		30: (*Spr.*)
			IF mcHeightMoveAbsolute.Done AND
				(mcScrewer1MoveRelative.Done OR NOT bOptionScrewingBackwardsInPushingPosition OR NOT bRun1) AND 	
				(mcScrewer2MoveRelative.Done OR NOT bOptionScrewingBackwardsInPushingPosition OR NOT bRun2) 	 			
			THEN	
				mcHeightMoveAbsolute.Execute					:=	FALSE;
				mcScrewer1MoveRelative.Execute					:=	FALSE;
				mcScrewer2MoveRelative.Execute					:=	FALSE;	
				iToPushingPositionCASE							:=	iToPushingPositionCASE	+	10;
			END_IF

		40:  (*Opcja - Dodatkowe zamknięcie chwytakiem przed zakręceniem *)
				IF bOptionCapPositioning AND sTool <> 'ksztaltowa/do kulek' AND sTool <> 'wbijajaca' THEN
					CASE iCloseGripperBeforeScrewingCASE OF
						0:
							bGripper1Actuator					:=	bRun1;
							bGripper2Actuator					:=	bRun2;
							iCloseGripperBeforeScrewingCASE		:=	iCloseGripperBeforeScrewingCASE	+10;
						10:	
							IF 	(tonGripper1Delay.Q OR NOT bRun1) AND 
								(tonGripper2Delay.Q OR NOT bRun2) 
							THEN					
								iCloseGripperBeforeScrewingCASE	:=	iCloseGripperBeforeScrewingCASE	+10;
							END_IF
						20:	
								bGripper1Actuator				:=	bGripper1Actuator	:=	FALSE;		
								iCloseGripperBeforeScrewingCASE	:=	iCloseGripperBeforeScrewingCASE	+10;
						30:
							IF 	(tonGripper1ReliseDelay2.Q OR NOT bRun1) AND 
								(tonGripper2ReliseDelay2.Q OR NOT bRun2) 
							THEN					
								iCloseGripperBeforeScrewingCASE	:=	iCloseGripperBeforeScrewingCASE	+10;
							END_IF
						40:
						
							iCloseGripperBeforeScrewingCASE		:=	0;
							iToPushingPositionCASE				:=	iToPushingPositionCASE	+	10;							
					END_CASE
				ELSE
					iToPushingPositionCASE						:=	iToPushingPositionCASE	+	10;
				END_IF

			
		50:	 (*Zamkniecie chwytaka i przejazd dalej*)
			IF sTool <> 'ksztaltowa/do kulek' AND sTool <> 'wbijajaca' THEN
				bGripper1Actuator								:=	bRun1;
				bGripper2Actuator								:=	bRun2;
			ELSE                                    	
				bGripper1Actuator								:=	FALSE;
				bGripper2Actuator								:=	FALSE;
			END_IF	

			IF bOptionOpenedGripperWhenFindingScrew AND bOptionFindScrewInPushingPosition THEN
				bGripper1Actuator								:=	FALSE;
				bGripper2Actuator								:=	FALSE;
			END_IF
			
			IF 	(tonGripper1Delay.Q OR sTool = 'ksztaltowa/do kulek' OR sTool = 'wbijajaca' OR bOptionOpenedGripperWhenFindingScrew AND bOptionFindScrewInPushingPosition OR NOT bRun1) AND 
				(tonGripper2Delay.Q OR sTool = 'ksztaltowa/do kulek' OR sTool = 'wbijajaca' OR bOptionOpenedGripperWhenFindingScrew AND bOptionFindScrewInPushingPosition OR NOT bRun2) 
			THEN
          		         	
				iToPushingPositionCASE							:=	iToPushingPositionCASE	+	10;
			END_IF	
		
				
		60:(*Opcja - Obrót z pozycji docisku do zakrecania *)
			IF bOptionFindScrewRotateFromPushingToScrewingSensor AND NOT bOptionFindScrewInPushingPosition THEN
				lrFindigScrewDegree								:=	180;	
			                                    				
				uiScrewing1TorqueControl						:=	6000;
				mcScrewer1MoveRelative.Velocity					:=	lrScrewerSpeed;		
				mcScrewer1MoveRelative.Execute					:=	bRun1;
							                    				
				uiScrewing2TorqueControl						:=	6000;
				mcScrewer2MoveRelative.Velocity					:=	lrScrewerSpeed;		
				mcScrewer2MoveRelative.Execute					:=	bRun2;
				iToPushingPositionCASE							:=	iToPushingPositionCASE	+	10;
				
			ELSE 
				iToPushingPositionCASE							:=	iToPushingPositionCASE	+	10;
			END_IF
				
		70:
		
			IF bOptionFindScrewInPushingPosition THEN
				eRunningState									:=	E_GripperScrewer.eFindingScrew;
			ELSE
				eRunningState									:=	E_GripperScrewer.eToScrewingPosition;
			END_IF
			
			iToPushingPositionCASE						:=	0;
	
				
		END_CASE
		
		(*w1
		bGripper1Actuator								:=	FALSE;
		bGripper2Actuator								:=	FALSE;
		mcHeightMoveAbsolute.Execute					:=	TRUE;
		mcHeightMoveAbsolute.Velocity					:=	lrHeightSpeed;
		mcHeightMoveAbsolute.Position					:=	lrHeightPushingPosition;

		(*Opcja - obrót do tyłu w momencie dojazdu do pozycji docisku*)
		IF bOptionScrewingBackwardsInPushingPosition THEN
			lrFindigScrewDegree				:=	180;	
			
			uiScrewing1TorqueControl		:=	6000;
			mcScrewer1MoveRelative.Velocity	:=	lrScrewerSpeed/2;		
			mcScrewer1MoveRelative.Execute	:=	bRun1;
			
			uiScrewing2TorqueControl		:=	6000;
			mcScrewer2MoveRelative.Velocity	:=	lrScrewerSpeed/2;		
			mcScrewer2MoveRelative.Execute	:=	bRun2;
		END_IF
	
		IF mcHeightMoveAbsolute.Done AND
			(mcScrewer1MoveRelative.Done OR NOT bOptionScrewingBackwardsInPushingPosition OR NOT bRun1) AND // Opcja
			(mcScrewer2MoveRelative.Done OR NOT bOptionScrewingBackwardsInPushingPosition OR NOT bRun2) 	 // Opcja			
		THEN		
			
			IF bOptionCapPositioning THEN //OPCJA. Dodatkowe zamknięcie chwytakiem przed zakręceniem (do testów)
				CASE iCloseGripperBeforeScrewingCASE OF
					0:
						IF iTool <> 2 THEN
							bGripper1Actuator						:=	bRun1;
							bGripper2Actuator						:=	bRun2;
						ELSE
							bGripper1Actuator						:=	FALSE;
							bGripper2Actuator						:=	FALSE;
						END_IF
						
						iCloseGripperBeforeScrewingCASE		:=	iCloseGripperBeforeScrewingCASE	+10;
						
					10:	
						IF iTool <> 2 THEN
							bGripper1Actuator						:=	bRun1;
							bGripper2Actuator						:=	bRun2;
						ELSE
							bGripper1Actuator						:=	FALSE;
							bGripper2Actuator						:=	FALSE;
						END_IF		
							
						IF (tonGripper1Delay.Q OR NOT bRun1) AND (tonGripper2Delay.Q OR NOT bRun2) THEN
							bGripper1Actuator						:=	bGripper1Actuator	:=	FALSE;							
							iCloseGripperBeforeScrewingCASE	:=	iCloseGripperBeforeScrewingCASE	+10;
						END_IF
					
					20:
						IF  tonGripper1ReliseDelay.Q AND tonGripper2ReliseDelay.Q THEN // Czas na otwarcie chwytaków
											
							mcHeightMoveAbsolute.Execute			:=	FALSE;
							eRunningState							:=	E_GripperScrewer.eToScrewingPosition;
							iCloseGripperBeforeScrewingCASE	:=	0;
						END_IF
													
				END_CASE

			ELSE
				IF iTool <> 2 THEN
					bGripper1Actuator					:=	bRun1;
					bGripper2Actuator					:=	bRun2;
				ELSE
					bGripper1Actuator					:=	FALSE;
					bGripper2Actuator					:=	FALSE;
				END_IF
									
				IF ((tonGripper1Delay.Q OR NOT bRun1) AND (tonGripper2Delay.Q OR NOT bRun2)) OR bOptionOpenedGripperWhenFindingScrew THEN
					mcHeightMoveAbsolute.Execute		:=	FALSE;
					mcScrewer1MoveRelative.Execute		:=	FALSE;
					mcScrewer2MoveRelative.Execute		:=	FALSE;
					
					IF bOptionFindScrewRotateFromPushingToScrewingSensor THEN
						lrFindigScrewDegree				:=	180;	
			
						uiScrewing1TorqueControl		:=	6000;
						mcScrewer1MoveRelative.Velocity	:=	lrScrewerSpeed;		
						mcScrewer1MoveRelative.Execute	:=	bRun1;
						
						uiScrewing2TorqueControl		:=	6000;
						mcScrewer2MoveRelative.Velocity	:=	lrScrewerSpeed;		
						mcScrewer2MoveRelative.Execute	:=	bRun2;
					END_IF
					
					IF	(mcScrewer1MoveRelative.Execute OR NOT bRun1 OR NOT bOptionFindScrewRotateFromPushingToScrewingSensor) AND
						(mcScrewer2MoveRelative.Execute OR NOT bRun2 OR NOT bOptionFindScrewRotateFromPushingToScrewingSensor) THEN
						eRunningState						:=	E_GripperScrewer.eToScrewingPosition;
					END_IF
					IF bOptionFindScrewInPushingPosition AND NOT bOptionFindScrewRotateFromPushingToScrewingSensor THEN //Opcja - szukanie gwintu w pozycji docisku
						IF 	bOptionOpenedGripperWhenFindingScrew THEN //Opcja - szukanie gwintu na otwartym chwytaku
							bGripper1Actuator				:=	FALSE;
							bGripper2Actuator				:=	FALSE;
						END_IF					
					
						eRunningState					:=	E_GripperScrewer.eFindingScrew;
					END_IF
					
				END_IF	
			END_IF
		END_IF
	*)
END_ACTION

ACTION Running5FindingScrew:
(*Opcja 1 Szukania gwintu - zwykłe szukanie*) 
IF NOT bOptionFindScrewWithHeightSensor THEN
	(*Opcja cofniecie o zadany kąt*)	
	CASE iFindingScrewCASE OF
				
			0:	// Czyszczenie
				mcScrewer1MoveRelative.Execute				:=	FALSE;
				mcScrewer2MoveRelative.Execute				:=	FALSE;		
				lrScrewer1MaxTorqueWhenFindingScrew			:=	0;
				lrScrewer2MaxTorqueWhenFindingScrew			:=	0;
				lrStartPosition1FindingScrew 				:=	Screwing1AxisRef.NcToPlc.ActPos;
				lrStartPosition2FindingScrew 				:=	Screwing2AxisRef.NcToPlc.ActPos;			
				uiScrewing1TorqueControl					:=	6000;
				uiScrewing2TorqueControl					:=	6000;			
				bScrew1Found								:=	FALSE;
				bScrew2Found								:=	FALSE;
				iFindingScrewCASE							:=	iFindingScrewCASE	+	10;
						
			10: (*ruch o zadany kat*)
				mcScrewer1MoveRelative.Velocity		:=	lrScrewerSpeed;
				mcScrewer1MoveRelative.Execute		:=	bRun1;
				
				mcScrewer2MoveRelative.Velocity		:=	lrScrewerSpeed;
				mcScrewer2MoveRelative.Execute		:=	bRun2;
				
				IF	(NOT bRun1 OR mcScrewer1MoveRelative.Done) AND
					(NOT bRun2 OR mcScrewer2MoveRelative.Done)
			
				THEN		
					lrScrewer1MaxTorqueWhenFindingScrew	:= 0;
					lrScrewer2MaxTorqueWhenFindingScrew	:= 0;
					mcScrewer1MoveRelative.Execute		:=	FALSE;
					mcScrewer1MoveRelative.Execute		:=	FALSE;
					iFindingScrewCASE					:=	iFindingScrewCASE	+	10;	
				END_IF
					
			20:
				lrStartPosition1						:=	Screwing1AxisRef.NcToPlc.ActPos;
				lrStartPosition2						:=	Screwing2AxisRef.NcToPlc.ActPos;
				iFindingScrewCASE 						:=	0;
				eRunningState							:=	E_GripperScrewer.eScrewing;
				IF bOptionFindScrewInPushingPosition THEN // Opcja - szukanie gwintu w pozycji docisku
					// Przejście do pozycji zakręcania, dlatego że był w pozycji docisku
					eRunningState							:=	E_GripperScrewer.eToScrewingPosition;
				END_IF
				IF NOT bHeightGearingWithScrewer THEN 	(* Wersja bez gearowania*)
					mcScrewer1MoveVelocity.Execute		:= bRun1;
					mcScrewer2MoveVelocity.Execute		:= bRun2;
					eRunningState:=E_GripperScrewer.eScrewing;
				ELSE 									(* Wersja z gearowaniem*)
					iFindingScrewCASE 						:=	0;
					eRunningState							:=	E_GripperScrewer.eScrewing;
					IF bOptionFindScrewInPushingPosition THEN // Opcja - szukanie gwintu w pozycji docisku
						// Przejście do pozycji zakręcania, dlatego że był w pozycji docisku
						eRunningState							:=	E_GripperScrewer.eToScrewingPosition;
					END_IF
				END_IF
	END_CASE

ELSE (*Opcja 2 Szukania gwintu - szukanie z czujnikiem wysokości*) 
		CASE iFindingScrewCASE OF
			
		0:	// Czyszczenie
			mcScrewer1MoveRelative.Execute				:=	FALSE;
			lrStartPosition1FindingScrew 				:=	Screwing1AxisRef.NcToPlc.ActPos;
			lrStartPosition2FindingScrew 				:=	Screwing2AxisRef.NcToPlc.ActPos;			
			uiScrewing1TorqueControl					:=	6000;
			uiScrewing2TorqueControl					:=	6000;			
			bScrew1Found								:=	FALSE;
			bScrew2Found								:=	FALSE;
			bScrew1MinFound								:=	FALSE;
			bScrew2MinFound								:=	FALSE;			
			lrScrewerMaxSensorHeightWhenFindingScrew	:=	-100000;
			lrScrewerMinSensorHeightWhenFindingScrew	:=	100000;
			iFindingScrewCASE							:=	iFindingScrewCASE	+	10;


		

			
		10: // Rozpoczęcie ruchu w tył i szukanie MAX wysokości oraz uskoku - początek gwintu
			


			uiScrewing1TorqueControl					:=	6000;
			mcScrewer1MoveRelative.Velocity				:=	lrScrewerSpeed;
			//Zabezpieczenie - jak za szybko się kręci to nie opada zakręcarka i nie łapie gwintu
			IF mcScrewer1MoveRelative.Velocity > 2400	THEN
				mcScrewer1MoveRelative.Velocity			:= 2400;
			END_IF	
			mcScrewer1MoveRelative.Execute				:=	bRun1;				
			IF lrScrewerMaxSensorHeightWhenFindingScrew<rSensorHeightCV  THEN
				lrScrewerMaxSensorHeightWhenFindingScrew:=	rSensorHeightCV;
			END_IF			
			//Jak znajdziemy uskok - to początek gwintu - uskok o 0.3 do 0.5 podziałki bo całego nie wykryje
			IF ((rSensorHeightCV+lrPackageThreadPitch*0.3)<lrScrewerMaxSensorHeightWhenFindingScrew) THEN //Było z krotnoscia gwintu ale tak ma wiekszy sens
				bScrew1Found							:=	TRUE;
				lrStartPosition1FindingScrew 			:=	Screwing1AxisRef.NcToPlc.ActPos; //Pozycja złapania gwintu
			END_IF
			//Koniec wyszukiwania - albo koniec ruchu albo znaleziony gwint
			IF (mcScrewer1MoveRelative.Done OR NOT bRun1) OR bScrew1Found THEN
				mcScrewer1MoveRelative.Execute			:=	FALSE;
				mcScrewer1Stop.Execute					:= TRUE;
			//	bFindScrewAdjustSensorHeight			:=	FALSE;	
			//	iFindScrewAdjustSensorHeight			:=	iFindScrewAdjustSensorHeight	+	1;
					
				iFindingScrewCASE						:=	iFindingScrewCASE	+	10;
			END_IF

			
		20: // Przejście dalej gdy jest gotowość
			IF NOT mcScrewer1MoveRelative.Busy AND NOT mcScrewer2MoveRelative.Busy AND mcScrewer1Stop.Done THEN
				mcScrewer1Stop.Execute					:= 	FALSE;			
				iFindingScrewCASE						:=	iFindingScrewCASE	+	10;	
			END_IF
			
		30://Koniec ruchu
			lrStartPosition1						:=	lrStartPosition1FindingScrew;
			lrStartPosition2						:=	Screwing2AxisRef.NcToPlc.ActPos;
			iFindingScrewCASE 						:=	0;
			eRunningState							:=	E_GripperScrewer.eScrewing;
			IF bOptionFindScrewInPushingPosition THEN // Opcja - szukanie gwintu w pozycji docisku
				// Przejście do pozycji zakręcania, dlatego że był w pozycji docisku
				eRunningState							:=	E_GripperScrewer.eToScrewingPosition;
			END_IF
		END_CASE	
			
//		10: // Rozpoczęcie ruchu w tył i szukanie MIN i MAX momentu
//			// Tylko 1 zakręcarka szuka Min i Max po każdej zmianie
//			// Uruchom szukanie jeżeli są wartości domyślne
//			IF lrScrewerMaxSensorHeightWhenFindingScrew = -100000 OR lrScrewerMinSensorHeightWhenFindingScrew = 100000 THEN
//				bFindScrewAdjustSensorHeight				:= TRUE;
//				lrScrewerMaxSensorHeightWhenFindingScrew	:=	-100000; //Musi być INIT -100000
//				lrScrewerMinSensorHeightWhenFindingScrew	:=	100000;
//			END_IF
			
//			IF bFindScrewAdjustSensorHeight THEN
//				uiScrewing1TorqueControl					:=	6000;
//				lrFindigScrewDegree							:=	720;
//				mcScrewer1MoveRelative.Velocity				:=	200;
//				mcScrewer1MoveRelative.Execute				:=	bRun1;
							
//				IF lrScrewerMaxSensorHeightWhenFindingScrew<diSensorHeightCV THEN
//					lrScrewerMaxSensorHeightWhenFindingScrew:=	diSensorHeightCV;
//				END_IF			
//				IF lrScrewerMinSensorHeightWhenFindingScrew>diSensorHeightCV THEN
//					lrScrewerMinSensorHeightWhenFindingScrew:=	diSensorHeightCV;
//				END_IF		
			
//				IF (mcScrewer1MoveRelative.Done OR NOT bRun1) THEN
//					mcScrewer1MoveRelative.Execute			:=	FALSE;
//					bFindScrewAdjustSensorHeight			:=	FALSE;	iFindScrewAdjustSensorHeight	:=	iFindScrewAdjustSensorHeight	+	1;
//					iFindingScrewCASE						:=	iFindingScrewCASE	+	10;
//				END_IF
//			ELSE
//				iFindingScrewCASE						:=	iFindingScrewCASE	+	10;
//			END_IF

			
//		30: // Rozpoczęcie szukanie największego momentu o określony maksymalny kąt
//			uiScrewing1TorqueControl					:=	6000;
//			mcScrewer1MoveRelative.Velocity				:=	500;//lrScrewerSpeed;///2;
//			mcScrewer1MoveRelative.Execute				:=	bRun1;
			
//			uiScrewing2TorqueControl					:=	6000;
//			mcScrewer2MoveRelative.Velocity				:=	500;//lrScrewerSpeed;///2;
//			mcScrewer2MoveRelative.Execute				:=	bRun2;		
	
//			iFindingScrewCASE							:=	iFindingScrewCASE	+	10;	
			
//		40:	//Szukanie określonego momentu po 200 st. i zatrzymanie ruchu 


//			(*Pierwsze szukanie*)
//			IF NOT bScrew1MinFound THEN															(*W1*)
//				IF ABS(ABS(lrStartPosition1FindingScrew)-ABS(Screwing1AxisRef.NcToPlc.ActPos))	>	100  THEN 
//					//IF lrScrewer1ActualTorque > (lrScrewer1MinTorqueWhenFindingScrew - 5) AND lrScrewer1ActualTorque < (lrScrewer1MaxTorqueWhenFindingScrew + 15) THEN		
////					IF diSensorHeightCV < -39000 THEN		(*W2*) //Dla Słoików 300ml
//					IF diSensorHeightCV < ((lrScrewerMaxSensorHeightWhenFindingScrew+lrScrewerMinSensorHeightWhenFindingScrew)/2) THEN		(*W2*) //Dla Słoików 300ml						
//						bScrew1MinFound						:=	TRUE;
//						lrStartPosition1FindingScrew 		:=	Screwing1AxisRef.NcToPlc.ActPos;
//					END_IF	
//				END_IF
//			END_IF
//			IF NOT bScrew2MinFound THEN															(*W1*)
//				IF ABS(ABS(lrStartPosition2FindingScrew)-ABS(Screwing2AxisRef.NcToPlc.ActPos))	>	100  THEN 
////					IF diSensorHeightCV < -39000 THEN		(*W2*)	//Dla Słoików 300ml	
//					IF diSensorHeightCV < ((lrScrewerMaxSensorHeightWhenFindingScrew+lrScrewerMinSensorHeightWhenFindingScrew)/2) THEN		(*W2*)	//Dla Słoików 300ml	
//						bScrew2MinFound						:=	TRUE;	
//						lrStartPosition2FindingScrew 		:=	Screwing2AxisRef.NcToPlc.ActPos;
//					END_IF	
//				END_IF	
//			END_IF
//			lrScrewerOffsetSensorHeightWhenFindingScrew	:=	((lrScrewerMaxSensorHeightWhenFindingScrew+lrScrewerMinSensorHeightWhenFindingScrew)/2)
//																+(lrScrewerMinSensorHeightWhenFindingScrew-lrScrewerMaxSensorHeightWhenFindingScrew)/6;
			
//			(*Drugie szukanie*)																					(*W3*)
//			IF bScrew1MinFound AND ABS(ABS(lrStartPosition1FindingScrew)-ABS(Screwing1AxisRef.NcToPlc.ActPos))	>	10  THEN 
				
//				IF diSensorHeightCV > lrScrewerOffsetSensorHeightWhenFindingScrew THEN		(*W4*)	//Dla Słoików 300ml
//					bScrew1Found						:=	TRUE;
//					mcScrewer1MoveRelative.Execute		:=	FALSE;
//					lrStartPosition1FindingScrew 		:=	Screwing1AxisRef.NcToPlc.ActPos;
//				END_IF
//			END_IF																								(*W3*)
//			IF bScrew2MinFound AND ABS(ABS(lrStartPosition2FindingScrew)-ABS(Screwing2AxisRef.NcToPlc.ActPos))	>	10  THEN 
//				IF diSensorHeightCV > ((lrScrewerMaxSensorHeightWhenFindingScrew+lrScrewerMinSensorHeightWhenFindingScrew)/2) THEN		(*W4*)	//Dla Słoików 300ml
//					bScrew2Found						:=	TRUE;
//					mcScrewer2MoveRelative.Execute		:=	FALSE;
//					lrStartPosition2FindingScrew 		:=	Screwing1AxisRef.NcToPlc.ActPos;
//				END_IF
//			END_IF

//			IF bScrew1Found  THEN

//				uiScrewing1TorqueControl		:=	6000;
//				mcScrewer1Stop.Execute			:=	TRUE;
				
//			END_IF
			
//			IF bScrew2Found  THEN

//				uiScrewing2TorqueControl		:=	6000;
//				mcScrewer2Stop.Execute			:=	TRUE;
//			END_IF			
			
//			IF	((bScrew1Found AND mcScrewer1Stop.Done) OR NOT bRun1 OR mcScrewer1MoveRelative.Done) AND
//				((bScrew2Found AND mcScrewer2Stop.Done) OR NOT bRun2 OR mcScrewer2MoveRelative.Done)
//			THEN
//				 mcScrewer1MoveRelative.Execute 	:=	FALSE;
//				 mcScrewer1Stop.Execute				:=	FALSE;
//				 mcScrewer2MoveRelative.Execute 	:=	FALSE;		
//				 mcScrewer2Stop.Execute				:=	FALSE;	 
//				 iFindingScrewCASE					:=	iFindingScrewCASE	+	10;	
//			END_IF
			
//		50: 
//			IF tonFindingScrewDelay.Q THEN
// 				iFindingScrewCASE					:=	iFindingScrewCASE	+	10;						
//			END_IF




END_IF
END_ACTION

ACTION Running6ScrewingMomentaryMode:
IF mcScrewer1TorqueControl.Error OR mcScrewer1MoveVelocity.Error OR mcScrewer1MoveVelocity2.Error
	 OR mcScrewer1MoveVelocity3.Error OR mcScrewer1MoveRelative.Error OR mcScrewer1MoveAbsolute.Error THEN
	bTest:= TRUE;
END_IF
tonInEndVelocity(IN:=mcScrewer1MoveContinuousRel.InEndVelocity, PT:=T#2MS);


				(********** TRYB MOMENTOWY **********)
					CASE iScrewingCase OF 	
					0:
						(* Wersja 2 - gearowanie Multi Master***************************************************************) 
						IF iTool <> 2 THEN
							bGripper1Actuator						:=	bRun1; // Ponowne załączanie chwytaków, dlatego
							bGripper2Actuator						:=	bRun2; // że jest możliwa duża ilość opcji
						ELSE
							bGripper1Actuator						:=	FALSE; // Ponowne załączanie chwytaków, dlatego
							bGripper2Actuator						:=	FALSE;
						END_IF
						//Właczenie sięcia osi
						mcHeightGearInMultiMaster.Enable			:=	TRUE;				
						//Jak osie spięte to początek kręcenia
						IF	mcHeightGearInMultiMaster.InGear AND 
							(tonGripper1Delay.Q OR sTool = 'ksztaltowa/do kulek' OR NOT bRun1) AND (tonGripper2Delay.Q OR sTool = 'ksztaltowa/do kulek'  OR NOT bRun2) // ton'y powinny być już wczesniej załączone jeżeli były chwytaki	
						THEN
							//Bloczek obrotu o zadany kąt i kontynuowania ruchu z zadaną prędkością
							mcScrewer1MoveContinuousRel.Execute				:= bRun1;
							//Kąt zmodyfikowany o różnicę między pozycją zatrzymania zakręcarki a pozycją wykrycia gwintu
							mcScrewer1MoveContinuousRel.Distance			:= Screwing1AxisRef.NcToPlc.ActPos - lrStartPosition1 + lrPackageTurnoversToFullScrewed*360.0-30.0;

							//DODAĆ ZABEZPIECZENIE JAK WYJDZIE ABSURDALNY KĄT
							
							//Prędkość na wyjściu z bloczka 120RPM - Inercja zakręcarki jest rozsądna
							mcScrewer1MoveContinuousRel.EndVelocity			:= 360*2;
							//Prędkość zakręcania wg parametrów
							mcScrewer1MoveContinuousRel.Velocity			:= (lrScrewerSpeed);
														
							iScrewingCase									:=	25;//iScrewingCase + 10;			
						END_IF
						
					10:	
					
						IF ABS(ABS(lrStartPosition1)-ABS(Screwing1AxisRef.NcToPlc.ActPos))>(lrPackageTurnoversToFullScrewed*360.0-90.0)  THEN 
							mcScrewer1MoveVelocity.Execute					:= FALSE;
							mcScrewer1MoveVelocity2.Execute					:= bRun1;
							mcScrewer1MoveVelocity2.Velocity				:= 360;
							uiScrewing1TorqueControl						:=	60000;
						//	mcScrewer1TorqueControl.Torque					:=	-5000;		
						//	mcScrewer1TorqueControl.TorqueRamp				:=	80000;	
							mcScrewer1TorqueControl.VelocityLimitHigh		:=	360;//(lrScrewerSpeed)/3.0;
							mcScrewer1TorqueControl.VelocityLimitLow		:=	-360;//-(lrScrewerSpeed)/3.0;
							iScrewingCase									:=	iScrewingCase + 10;	
						END_IF	
							
//						IF ABS(ABS(lrStartPosition2)-ABS(Screwing2AxisRef.NcToPlc.ActPos))>(lrPackageTurnoversToFullScrewed*360.0/7)  THEN 
//							mcScrewer2TorqueControl.Torque					:=	-9;		
//							mcScrewer2TorqueControl.TorqueRamp				:=	1500;					
//							mcScrewer2TorqueControl.VelocityLimitLow		:=	-4000;
//						END_IF	
					20:	
						mcScrewer1MoveVelocity2.Execute					:= FALSE;
						IF ABS(ABS(lrStartPosition1)-ABS(Screwing1AxisRef.NcToPlc.ActPos))>(lrPackageTurnoversToFullScrewed*360.0-15.0)  THEN
							mcScrewer1MoveVelocity2.Execute					:= FALSE;
							mcScrewer1TorqueControl.Execute					:=	bRun1;
							mcScrewer1TorqueControl.Torque					:=	(INT_TO_UINT(iScrewer1SetTorque)+iScrewer1AddTorque);		
						//	mcScrewer1TorqueControl.TorqueRamp				:=	4000;					
						//	mcScrewer1TorqueControl.VelocityLimitLow		:=	- 10;//(lrScrewerSpeed)/3.0;
							iScrewingCase									:=	iScrewingCase + 10;	
						END_IF	
							
						IF ABS(ABS(lrStartPosition2)-ABS(Screwing2AxisRef.NcToPlc.ActPos))>(lrPackageTurnoversToFullScrewed*360.0/6)  THEN 
							mcScrewer2TorqueControl.Torque					:=	(INT_TO_UINT(iScrewer2SetTorque)+iScrewer2AddTorque);		
							mcScrewer2TorqueControl.TorqueRamp				:=	4000;					
							mcScrewer2TorqueControl.VelocityLimitLow		:=	-(lrScrewerSpeed);
						END_IF	
						
					25:
						//Jak dojedzie do końca ruchu
						IF mcScrewer1MoveContinuousRel.InEndVelocity AND tonInEndVelocity.Q THEN
							mcScrewer1MoveContinuousRel.Execute				:= FALSE;
							//Przygotowanie trybu momentowego
							mcScrewer1TorqueControl.Execute					:=	bRun1;
							mcScrewer1TorqueControl.Torque					:=	(INT_TO_UINT(iScrewer1SetTorque)+iScrewer1AddTorque);	
							mcScrewer1TorqueControl.TorqueRamp				:=	8000;
							mcScrewer1TorqueControl.VelocityLimitHigh		:=	360*2;//(lrScrewerSpeed)/3.0;
							mcScrewer1TorqueControl.VelocityLimitLow		:=	-360*2;//-(lrScrewerSpeed)/3.0;	
							iScrewingCase									:=	30;//iScrewingCase + 10;	
						END_IF
	
					30:
						IF tonMomentaryScrewing1Timer.Q OR bWarning1 THEN
							mcScrewer1Stop.Execute				:=	TRUE;
							bGripper1Actuator					:=	FALSE;
							mcScrewer1TorqueControl.Execute		:=	FALSE;
							uiScrewing1TorqueControl			:=	0;
							bScrewed1							:=	TRUE;	
						END_IF
						IF tonMomentaryScrewing2Timer.Q OR bWarning2 THEN
							mcScrewer2Stop.Execute				:=	TRUE;
							bGripper2Actuator					:=	FALSE;
							mcScrewer2TorqueControl.Execute		:=	FALSE;
							uiScrewing2TorqueControl			:=	0;
							bScrewed2							:=	TRUE;		
						END_IF
				
						// Warunki zakręcenia zaleznie od uruchomionej zakręcarki
						IF (bScrewed1 OR NOT bRun1) AND (bScrewed2 OR NOT bRun2) AND
							(mcScrewer1Stop.Done OR NOT mcScrewer1Stop.Execute) AND 
							(mcScrewer2Stop.Done OR NOT mcScrewer2Stop.Execute) THEN
								mcScrewer1Stop.Execute			:= FALSE;
								mcScrewer2Stop.Execute			:= FALSE;
								iScrewingCase					:= iScrewingCase + 10;		
						END_IF
					40:
						(* Rozgearowanie osi *)
						mcHeightGearOut.Execute				:=	TRUE;
						mcHeightGearInMultiMaster.Enable	:=	FALSE;
	
						IF  mcHeightGearOut.Done THEN
							mcHeightGearOut.Execute					:= FALSE;
							eRunningState							:= E_GripperScrewer.eHolding;	
							iScrewingCase							:= 0;	
						END_IF			
					END_CASE
END_ACTION

ACTION Running6ScrewingPositionTorqueMode:
				(********* TRYB POZYCYJNY  *********)
				
				lrPackageThreadPitch;	
				(*Wymuszanie zwiększonego momentu przez 1/4 całego zakręcania*)
				IF ABS(ABS(lrStartPosition1)-ABS(Screwing1AxisRef.NcToPlc.ActPos))>(lrPackageTurnoversToFullScrewed*360.0/7)  THEN 
							uiScrewing1TorqueControl			:=	(INT_TO_UINT(iScrewer1SetTorque+3)*10)+(iScrewer1AddTorque*10);	
				ELSE		uiScrewing1TorqueControl			:=	6000;
				END_IF
				//uiScrewing1TorqueControl			:=	(INT_TO_UINT(iScrewerSetTorque+3)*10)+iScrewer1AddTorque;	
				(*Wymuszanie zwiększonego momentu przez 1/4 całego zakręcania*)
				IF ABS(ABS(lrStartPosition2)-ABS(Screwing2AxisRef.NcToPlc.ActPos))>(lrPackageTurnoversToFullScrewed*360.0/7)  THEN 
							uiScrewing2TorqueControl			:=	(INT_TO_UINT(iScrewer2SetTorque+3)*10)+(iScrewer2AddTorque*10);		
				ELSE		uiScrewing2TorqueControl			:=	6000;
				END_IF	

					CASE iScrewingCase OF 	
					0:
						(* Wersja 2 - gearowanie Multi Master***************************************************************) 
						IF iTool <> 2 THEN
							bGripper1Actuator						:=	bRun1; // Ponowne załączanie chwytaków, dlatego
							bGripper2Actuator						:=	bRun2; // że jest możliwa duża ilość opcji
						ELSE
							bGripper1Actuator						:=	FALSE; // Ponowne załączanie chwytaków, dlatego
							bGripper2Actuator						:=	FALSE; // że jest możliwa duża ilość opcji
						END_IF
						mcHeightGearInMultiMaster.Enable			:=	TRUE;				
						(* Start zakręcania *)
						IF	mcHeightGearInMultiMaster.InGear AND 
							(tonGripper1Delay.Q OR sTool = 'ksztaltowa/do kulek' OR NOT bRun1) AND (tonGripper2Delay.Q OR sTool = 'ksztaltowa/do kulek' OR NOT bRun2) // ton'y powinny być już wczesniej załączone jeżeli były chwytaki	
						THEN

							CASE iScrewing2Case OF 	
								
							0:
							
								mcScrewer1MoveVelocity2.Velocity		:=	5000;
								mcScrewer1MoveVelocity2.Execute		:=	bRun1;
								mcScrewer1MoveVelocity2.Direction	:=	MC_Positive_Direction;
																				
								mcScrewer2MoveVelocity2.Velocity		:=	5000;
								mcScrewer2MoveVelocity2.Execute		:=	bRun2;
								mcScrewer2MoveVelocity2.Direction	:=	MC_Positive_Direction;	
	
								iScrewing2Case						:=	iScrewing2Case + 10;										
							
							10:
								mcScrewer1MoveVelocity2.Execute		:=	FALSE;
								mcScrewer2MoveVelocity2.Execute		:=	FALSE;
							
								iScrewing2Case						:=	iScrewing2Case + 10;
	
							20:
							
								mcScrewer1MoveVelocity.Velocity		:=	lrScrewerSpeed;		
								mcScrewer1MoveVelocity.Direction	:=	MC_Positive_Direction;	
								IF ABS(ABS(lrStartPosition1)-ABS(Screwing1AxisRef.NcToPlc.ActPos))>(lrPackageTurnoversToFullScrewed*360.0/7)  THEN 									
									mcScrewer1MoveVelocity.Execute		:=	bRun1;									
								END_IF
								mcScrewer2MoveVelocity.Velocity		:=	lrScrewerSpeed;	
								mcScrewer1MoveVelocity.Direction		:=	MC_Positive_Direction;	
								IF ABS(ABS(lrStartPosition2)-ABS(Screwing2AxisRef.NcToPlc.ActPos))>(lrPackageTurnoversToFullScrewed*360.0/7)  THEN 
	
									mcScrewer2MoveVelocity.Execute		:=	bRun2;
								END_IF			

								IF (mcScrewer1MoveVelocity.Execute OR NOT bRun1) AND (mcScrewer2MoveVelocity.Execute OR NOT bRun2) THEN
									iScrewing2Case					:= 0	;
									iScrewingCase					:= iScrewingCase + 10;		
								END_IF
								
							END_CASE
							
						END_IF
						
					10:	
					
						(*Zmniejszanie prędkości jeżeli jest już przytrzymanie*)
						IF tonTightScrewing1Timer.ET > T#0S AND Screwing1AxisRef.NcToPlc.ActVelo < 10 THEN
							//mcScrewer1MoveVelocity.Execute		:= FALSE;
							//mcScrewer1MoveVelocity2.Execute		:= FALSE;
							
							//mcScrewer1MoveVelocity3.Velocity	:=	10;
							//mcScrewer1MoveVelocity3.Execute		:=	bRun1;
							//mcScrewer1MoveVelocity3.Direction	:=	MC_Positive_Direction;		

							rScrewing1ProportionalGain	:= 0;
							//rScrewing2ProportionalGain	:= 0;												
						END_IF
						
						IF tonTightScrewing2Timer.ET > T#0S AND Screwing2AxisRef.NcToPlc.ActVelo < 10 THEN
							//mcScrewer2MoveVelocity.Execute		:= FALSE;
							//mcScrewer2MoveVelocity2.Execute		:= FALSE;
							
							//mcScrewer2MoveVelocity3.Velocity	:=	10;
							//mcScrewer2MoveVelocity3.Execute		:=	bRun1;
							//mcScrewer2MoveVelocity3.Direction	:=	MC_Positive_Direction;		

							//rScrewing1ProportionalGain	:= 0;
							rScrewing2ProportionalGain	:= 0;												
						END_IF					
					
						(* Sprawdzanie czy osiągnięto moment lub zbyt długie zakracanie*)				
						IF tonTightScrewing1Timer.Q OR bWarning1 THEN
							bGripper1Actuator					:=	FALSE;
							bScrewed1							:=	TRUE;	
						END_IF
						IF tonTightScrewing2Timer.Q OR bWarning2 THEN
							bGripper2Actuator					:=	FALSE;
							bScrewed2							:=	TRUE;		
						END_IF
	
						IF tonTightScrewing1TimerAndOpenedGripper.Q THEN
							mcScrewer1Stop.Execute				:=	TRUE;
							mcScrewer1MoveVelocity.Execute		:=	FALSE;
							mcScrewer1MoveVelocity2.Execute		:=	FALSE;
							mcScrewer1MoveVelocity3.Execute		:=	FALSE;							
							uiScrewing1TorqueControl			:=	0;
						END_IF
						IF tonTightScrewing2TimerAndOpenedGripper.Q THEN
							mcScrewer2Stop.Execute				:=	TRUE;
							mcScrewer2MoveVelocity.Execute		:=	FALSE;
							mcScrewer2MoveVelocity2.Execute		:=	FALSE;	
							mcScrewer2MoveVelocity3.Execute		:=	FALSE;							
							uiScrewing2TorqueControl			:=	0;
						END_IF
					
						// Warunki zakręcenia zaleznie od uruchomionej zakręcarki
						IF (tonTightScrewing1TimerAndOpenedGripper.Q OR NOT bRun1) AND (tonTightScrewing2TimerAndOpenedGripper.Q OR NOT bRun2) AND
							(mcScrewer1Stop.Done OR NOT mcScrewer1Stop.Execute) AND 
							(mcScrewer2Stop.Done OR NOT mcScrewer2Stop.Execute) THEN
								mcScrewer1Stop.Execute			:= FALSE;
								mcScrewer2Stop.Execute			:= FALSE;
								iScrewingCase					:= iScrewingCase + 10;		
						END_IF
						
					20:
						(* Rozgearowanie osi *)
						mcHeightGearOut.Execute				:=	TRUE;
						mcHeightGearInMultiMaster.Enable	:=	FALSE;
	
						IF  mcHeightGearOut.Done THEN
							mcHeightGearOut.Execute					:= FALSE;
							eRunningState							:= E_GripperScrewer.eHolding;	
							iScrewingCase							:= 0;	
						END_IF			
					END_CASE
END_ACTION

ACTION Screwer1ControlBlocks:
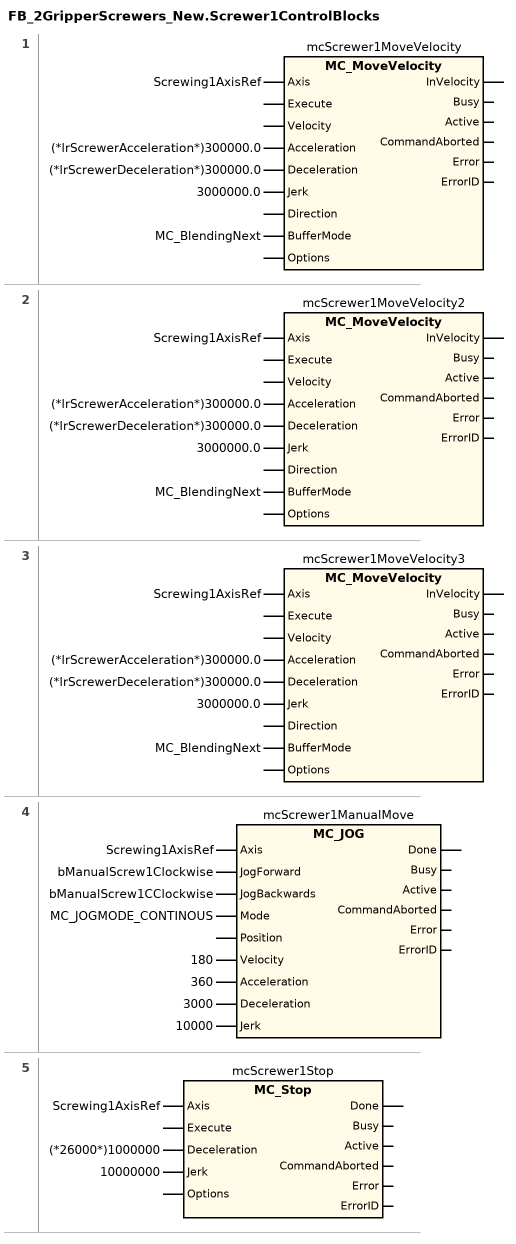
// NETWORK 1
mcScrewer1MoveVelocity(
    Axis := Screwing1AxisRef,
    Acceleration := (*lrScrewerAcceleration*)300000.0,
    Deceleration := (*lrScrewerDeceleration*)300000.0,
    Jerk := 3000000.0,
    BufferMode := MC_BlendingNext); // MC_MoveVelocity

// NETWORK 2
mcScrewer1MoveVelocity2(
    Axis := Screwing1AxisRef,
    Acceleration := (*lrScrewerAcceleration*)300000.0,
    Deceleration := (*lrScrewerDeceleration*)300000.0,
    Jerk := 3000000.0,
    BufferMode := MC_BlendingNext); // MC_MoveVelocity

// NETWORK 3
mcScrewer1MoveVelocity3(
    Axis := Screwing1AxisRef,
    Acceleration := (*lrScrewerAcceleration*)300000.0,
    Deceleration := (*lrScrewerDeceleration*)300000.0,
    Jerk := 3000000.0,
    BufferMode := MC_BlendingNext); // MC_MoveVelocity

// NETWORK 4
mcScrewer1ManualMove(
    Axis := Screwing1AxisRef,
    JogForward := bManualScrew1Clockwise,
    JogBackwards := bManualScrew1CClockwise,
    Mode := MC_JOGMODE_CONTINOUS,
    Velocity := 180,
    Acceleration := 360,
    Deceleration := 3000,
    Jerk := 10000); // MC_JOG

// NETWORK 5
mcScrewer1Stop(Axis := Screwing1AxisRef, Deceleration := (*26000*)1000000, Jerk := 10000000); // MC_Stop

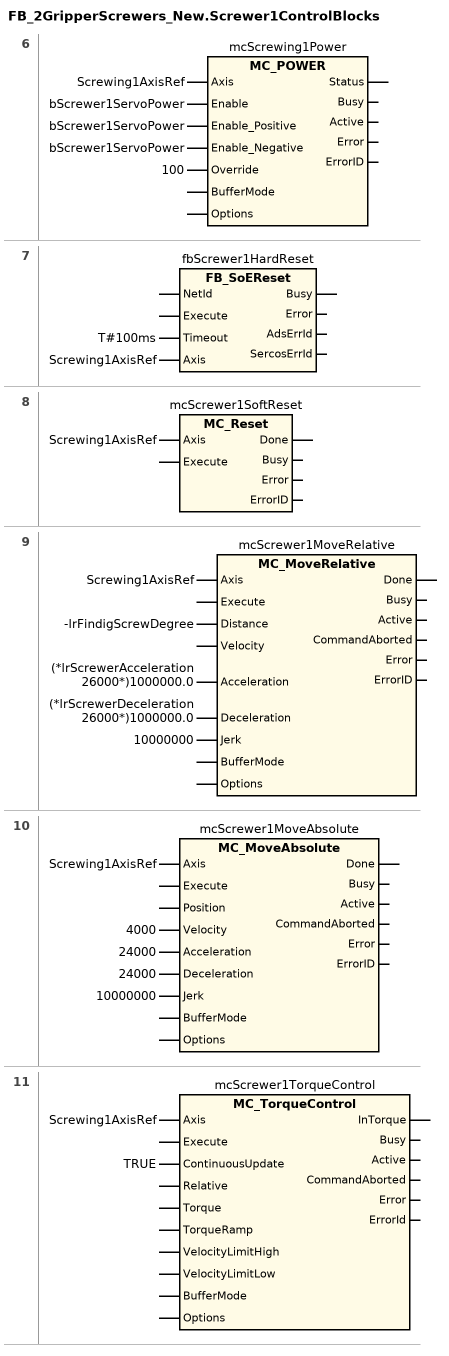
// NETWORK 6
mcScrewing1Power(
    Axis := Screwing1AxisRef,
    Enable := bScrewer1ServoPower,
    Enable_Positive := bScrewer1ServoPower,
    Enable_Negative := bScrewer1ServoPower,
    Override := 100); // MC_POWER

// NETWORK 7
fbScrewer1HardReset(Timeout := T#100ms, Axis := Screwing1AxisRef); // FB_SoEReset

// NETWORK 8
mcScrewer1SoftReset(Axis := Screwing1AxisRef); // MC_Reset

// NETWORK 9
mcScrewer1MoveRelative(
    Axis := Screwing1AxisRef,
    Distance := -lrFindigScrewDegree,
    Acceleration := (*lrScrewerAcceleration 26000*)1000000.0,
    Deceleration := (*lrScrewerDeceleration 26000*)1000000.0,
    Jerk := 10000000); // MC_MoveRelative

// NETWORK 10
mcScrewer1MoveAbsolute(
    Axis := Screwing1AxisRef,
    Velocity := 4000,
    Acceleration := 24000,
    Deceleration := 24000,
    Jerk := 10000000); // MC_MoveAbsolute

// NETWORK 11
mcScrewer1TorqueControl(Axis := Screwing1AxisRef, ContinuousUpdate := TRUE); // MC_TorqueControl

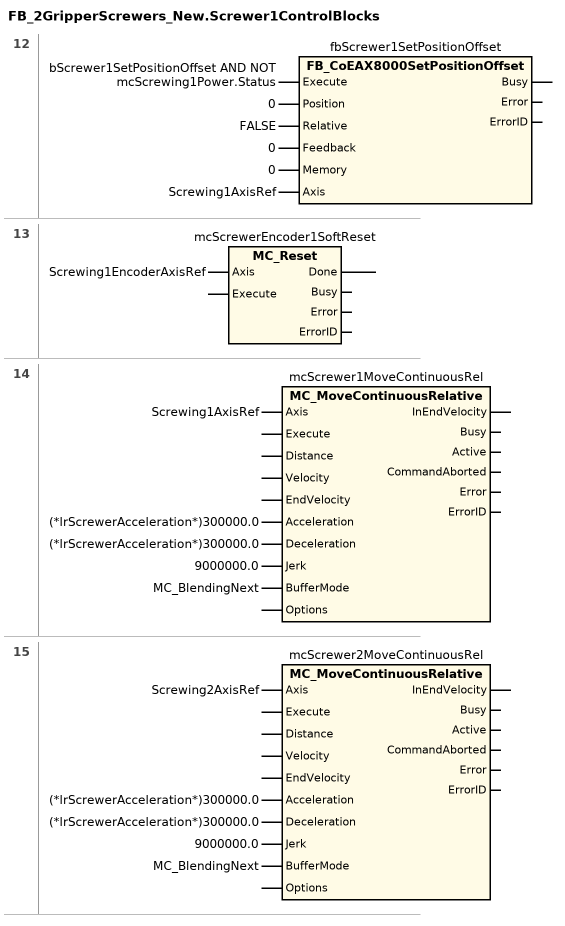
// NETWORK 12
fbScrewer1SetPositionOffset(
    Execute := bScrewer1SetPositionOffset AND NOT mcScrewing1Power.Status,
    Position := 0,
    Relative := FALSE,
    Feedback := 0,
    Memory := 0,
    Axis := Screwing1AxisRef); // FB_CoEAX8000SetPositionOffset

// NETWORK 13
mcScrewerEncoder1SoftReset(Axis := Screwing1EncoderAxisRef); // MC_Reset

// NETWORK 14
mcScrewer1MoveContinuousRel(
    Axis := Screwing1AxisRef,
    Acceleration := (*lrScrewerAcceleration*)300000.0,
    Deceleration := (*lrScrewerAcceleration*)300000.0,
    Jerk := 9000000.0,
    BufferMode := MC_BlendingNext); // MC_MoveContinuousRelative

// NETWORK 15
mcScrewer2MoveContinuousRel(
    Axis := Screwing2AxisRef,
    Acceleration := (*lrScrewerAcceleration*)300000.0,
    Deceleration := (*lrScrewerAcceleration*)300000.0,
    Jerk := 9000000.0,
    BufferMode := MC_BlendingNext); // MC_MoveContinuousRelative
END_ACTION

ACTION Screwer2ControlBlocks:
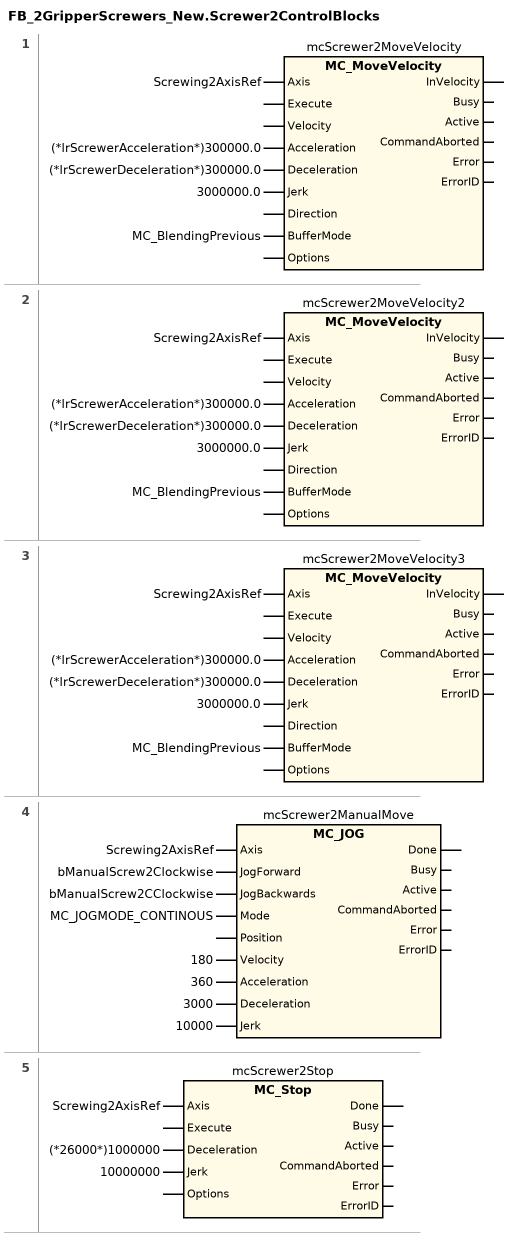
// NETWORK 1
mcScrewer2MoveVelocity(
    Axis := Screwing2AxisRef,
    Acceleration := (*lrScrewerAcceleration*)300000.0,
    Deceleration := (*lrScrewerDeceleration*)300000.0,
    Jerk := 3000000.0,
    BufferMode := MC_BlendingPrevious); // MC_MoveVelocity

// NETWORK 2
mcScrewer2MoveVelocity2(
    Axis := Screwing2AxisRef,
    Acceleration := (*lrScrewerAcceleration*)300000.0,
    Deceleration := (*lrScrewerDeceleration*)300000.0,
    Jerk := 3000000.0,
    BufferMode := MC_BlendingPrevious); // MC_MoveVelocity

// NETWORK 3
mcScrewer2MoveVelocity3(
    Axis := Screwing2AxisRef,
    Acceleration := (*lrScrewerAcceleration*)300000.0,
    Deceleration := (*lrScrewerDeceleration*)300000.0,
    Jerk := 3000000.0,
    BufferMode := MC_BlendingPrevious); // MC_MoveVelocity

// NETWORK 4
mcScrewer2ManualMove(
    Axis := Screwing2AxisRef,
    JogForward := bManualScrew2Clockwise,
    JogBackwards := bManualScrew2CClockwise,
    Mode := MC_JOGMODE_CONTINOUS,
    Velocity := 180,
    Acceleration := 360,
    Deceleration := 3000,
    Jerk := 10000); // MC_JOG

// NETWORK 5
mcScrewer2Stop(Axis := Screwing2AxisRef, Deceleration := (*26000*)1000000, Jerk := 10000000); // MC_Stop

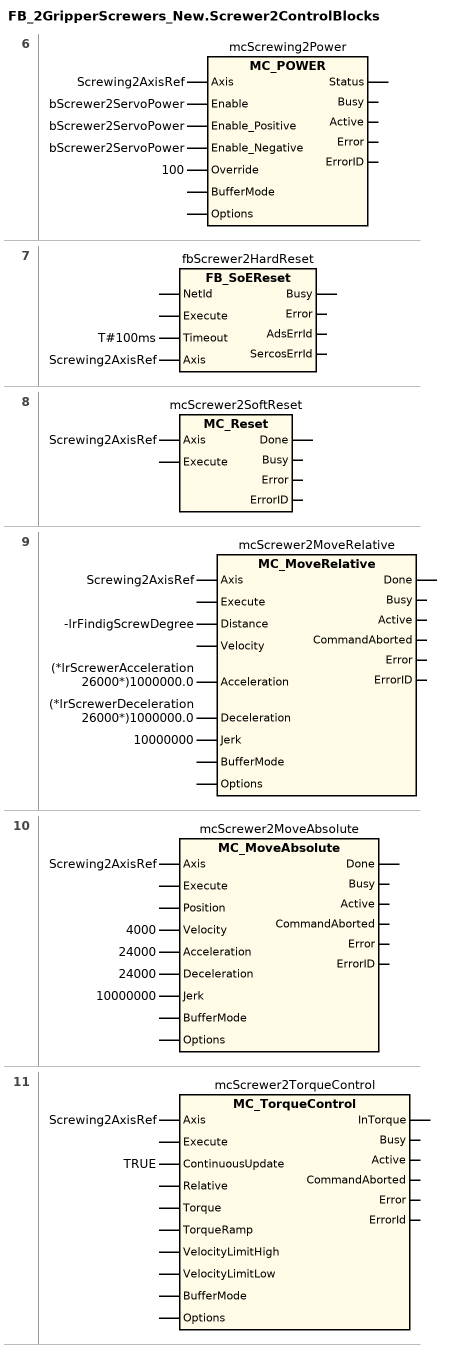
// NETWORK 6
mcScrewing2Power(
    Axis := Screwing2AxisRef,
    Enable := bScrewer2ServoPower,
    Enable_Positive := bScrewer2ServoPower,
    Enable_Negative := bScrewer2ServoPower,
    Override := 100); // MC_POWER

// NETWORK 7
fbScrewer2HardReset(Timeout := T#100ms, Axis := Screwing2AxisRef); // FB_SoEReset

// NETWORK 8
mcScrewer2SoftReset(Axis := Screwing2AxisRef); // MC_Reset

// NETWORK 9
mcScrewer2MoveRelative(
    Axis := Screwing2AxisRef,
    Distance := -lrFindigScrewDegree,
    Acceleration := (*lrScrewerAcceleration 26000*)1000000.0,
    Deceleration := (*lrScrewerDeceleration 26000*)1000000.0,
    Jerk := 10000000); // MC_MoveRelative

// NETWORK 10
mcScrewer2MoveAbsolute(
    Axis := Screwing2AxisRef,
    Velocity := 4000,
    Acceleration := 24000,
    Deceleration := 24000,
    Jerk := 10000000); // MC_MoveAbsolute

// NETWORK 11
mcScrewer2TorqueControl(Axis := Screwing2AxisRef, ContinuousUpdate := TRUE); // MC_TorqueControl

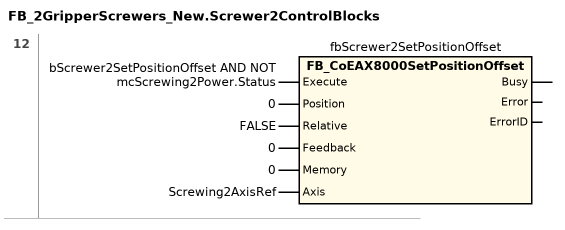
// NETWORK 12
fbScrewer2SetPositionOffset(
    Execute := bScrewer2SetPositionOffset AND NOT mcScrewing2Power.Status,
    Position := 0,
    Relative := FALSE,
    Feedback := 0,
    Memory := 0,
    Axis := Screwing2AxisRef); // FB_CoEAX8000SetPositionOffset
END_ACTION

ACTION Simulation:
(* Przyśpieszanie bloku gdy jest włączona symulacja*)

//tonSimulationScrewing1			(IN:=eRunningState=E_GripperScrewer.eScrewing 	AND bRun1 AND NOT bScrewed1 AND bSimulation,	PT:=T#0MS);
//tonSimulationScrewing2			(IN:=eRunningState=E_GripperScrewer.eScrewing 	AND bRun1 AND NOT bScrewed2 AND bSimulation,	PT:=T#0MS);

IF bSimulation THEN 			// Włączona symulacja
	tTooLongScrewing1 := T#250MS;
	tTooLongScrewing2 := T#250MS;	
ELSE							// Normalna praca
	tTooLongScrewing1 := T#2S; 	//Zmienić na 2
	tTooLongScrewing2 := T#2S;	//Zmienić na 2
END_IF
END_ACTION

ACTION Statistics:

IF LREAL_TO_INT(lrHeightEndScrewingPosition)<> LREAL_TO_INT(lrHeightReadyPosition) THEN
	rtrigCycleTimerRead(CLK:=LREAL_TO_INT(lrHeightActualPosition) = LREAL_TO_INT(lrHeightReadyPosition));
	IF rtrigCycleTimerRead.Q THEN
			tCycleTime:=tonCycleTimer.ET;
	END_IF
	tonCycleTimer(IN:=LREAL_TO_INT(lrHeightActualPosition) <> LREAL_TO_INT(lrHeightReadyPosition),PT:=T#1D);	
ELSE
	rtrigCycleTimerRead(CLK:=(eRunningState=E_GripperScrewer.eDone) OR (eRunningState=E_GripperScrewer.eNotDone));
	IF rtrigCycleTimerRead.Q THEN
		tCycleTime:=tonCycleTimer.ET;
	END_IF
	tonCycleTimer(IN:=eRunningState>E_GripperScrewer.eReady,PT:=T#1D);
END_IF
END_ACTION

ACTION Tools:
(*Narzędzia*)
AsToolDescription[0] := 'Głowica dwuszczękowa';
AsToolDescription[1] := 'Głowica trójszczękowa'; 
AsToolDescription[2] := 'Głowica kształtowa/do kulek';
AsToolDescription[3] := 'Głowica wbijająca'; 
AsToolDescription[4] := 'Głowica zasysająca';


(*Głowica wbijająca*)
IF iTool = 3 THEN
	bOptionCapPushingWithoutScrewing := TRUE;
ELSE
	bOptionCapPushingWithoutScrewing := FALSE;
END_IF

(*Przepisanie wybranego narzędzia do zmiennej typu string*)
(*!!!!! NIE ZMIENIAĆ OPISÓW, POWIĄZANE W PROGRAMIE !!!!!!*)
IF iTool = 0 THEN sTool := 'dwuszczekowa';			END_IF 
IF iTool = 1 THEN sTool := 'trojszczekowa';			END_IF
IF iTool = 2 THEN sTool := 'ksztaltowa/do kulek';	END_IF
IF iTool = 3 THEN sTool := 'wbijajaca';				END_IF
IF iTool = 4 THEN sTool := 'zasysajaca';			END_IF
END_ACTION

ACTION TorqueControl:

(*Konfiguracja MC_TorqueControl*)
//T_TorqueControlOptions;
mcScrewer1TorqueControl.Options.EnableManualTorqueStartValue := FALSE;//TRUE;
mcScrewer1TorqueControl.Options.ManualTorqueStartValue       := Screwing1AxisRef.NcToPlc.ActTorque;

mcScrewer2TorqueControl.Options.EnableManualTorqueStartValue := TRUE;
mcScrewer2TorqueControl.Options.ManualTorqueStartValue       :=  Screwing2AxisRef.NcToPlc.ActTorque;
END_ACTION

ACTION Warnings:
//Resetowanie warningów przy nastepnym cyklu

IF rtRun1.Q  OR rtRun2.Q THEN
	
	bWarning1			:=	FALSE;
	bWarning1A			:=	FALSE;
	bWarning1B			:=	FALSE;
	bWarning1C			:=	FALSE;
	bWarning1D			:=	FALSE;
	bWarning1E			:=	FALSE;	
	bWarning2			:=	FALSE;
	bWarning2A			:=	FALSE;
	bWarning2B			:=	FALSE;
	bWarning2C			:=	FALSE;
	bWarning2D			:=	FALSE;
	bWarning2E			:=	FALSE;
	udiWarningID		:=	0;
	sWarningDescription	:=	'';
END_IF
END_ACTION

END_FUNCTION_BLOCK

(* stored: Version 1.1.0.1, ProductVersion 3.1.4026.13, FileIdentifier 049f62b842b5e1f654cefd41391f1a267d8f2fbd, FileSignature 3e7d791a241618ec519fb3412899222f8602e77ce7a8cb2218fc0a6c49669b9543416119373265bfa7b2d214a8e4647ccf949d84cbebe9aa824864865ef52edb9322003cb9d9c3b3505495b8e606fb4507b7b841d78f7197b14acb816f192b69f2d59f298b65b5bfb9c38ac7fea521352669fa8406ee3c513c71c1b34259a5e6da06ed0a7b4bfc46f491fe3da6a9a96f84d0e225717740dcea9cc9ef6cbb1125f34fccba2f4b880716ac2844c92b99b917767408a5722cbe5e75eb287890ddfaad512cbd74b7ee89e224d84715a6093c677d1e4881b0d43163f381c14715acffb710de84d7497752697013e0434d818ba5d0bb4530b537d266eda15603c16633
   POU FB_2GripperScrewers_New: Id {b4fcfdb0-083b-4c26-b766-7363e9f32dbf}, SpecialFunc None
   Folder Methods: Id {bd8de6a0-2cfd-48d5-906c-fc91f347fbf7}
   Action AdjustingTorque: Id {ebc04306-77c2-4b14-baa7-efcee67b6099}
   Action aStationID: Id {df026cf7-8324-4d02-ae3a-044edb8f47cc}
   Action Control: Id {aa760fe9-b92d-4948-8caa-16ac2e81b340}
   Action ErrorHandling: Id {74b92e08-0fc6-4060-9784-f818a4b469a1}
   Action HeightControlBlocks: Id {040caa86-b824-4b62-8af6-db749774b2bc}
   Action Homing: Id {2f69e65e-c04e-4513-8137-7a6e094f7160}
   Action Limits: Id {2c71db91-320c-4d04-bc96-9439c1d329c0}
   Method M_PrepareToReady: Id {20a1ce0b-2a2d-4a67-a807-e9654d9c6b0b}
   Action ManualMovements: Id {d94f9ca6-587b-4ead-b37f-57d4afc50e3b}
   Action ManualMovementsStepMode: Id {dc1772fa-812a-4fd4-8512-79fa79ff1b94}
   Action ReadScrewingTorque: Id {26b2b602-bdb8-444a-8dac-028cf76735bf}
   Action ResetCommands: Id {f47b040e-729f-4e1f-a37a-2fc6ca6975a3}
   Action Running: Id {3f297f70-d94c-494b-a9ca-3e1d1f381b88}
   Action Running2ToPushingPosition: Id {6974bb38-9842-4112-a04a-40a8dc8dc7ca}
   Action Running5FindingScrew: Id {072135cd-dba2-431b-93e0-e70145258762}
   Action Running6ScrewingMomentaryMode: Id {cef86e03-c378-4354-9232-342573c49138}
   Action Running6ScrewingPositionTorqueMode: Id {a2d12478-e930-4110-9859-0a5b21d74693}
   Action Screwer1ControlBlocks: Id {fd1420bd-c5c7-49d1-8c0d-f35e35c9a9b9}
   Action Screwer2ControlBlocks: Id {fd4ed05f-9255-4e5c-8101-c7175ed6cf81}
   Action Simulation: Id {18b30540-2376-41d0-8cc6-802471651668}
   Action Statistics: Id {80798a50-95d5-4254-9f3c-af6cc198e53c}
   Action Tools: Id {4288a769-e8e3-41ed-a289-eae35581308a}
   Action TorqueControl: Id {f8728233-b731-448d-aedd-62ce54b7b1c2}
   Action Warnings: Id {5029350e-ab90-4e9e-8a89-79d867e9b6ff} *)
